FUNCTION_BLOCK FB_FlowLine
(*
********************************************************************************
* Name: FB_Camera
*
* Author:  AutomanH
* Version: 1.0.0
*
* Description:
*	Flow Line Program and motor control
*
* Remarks:
*
*
* Revisions:
*   V1.0.0 -Automanh 2022.06.08
* 	V1.1.0-Automanh 2022.06.20,Add ACT_Motor();
*		V2.0.0-Automanh 2022.07.18 add timeout alarm 
*********************************************************************************)
VAR_INPUT
 arIReachedSensor:ARRAY[1..iColumnsNum] OF BOOL;
 arIVTCCylHPSensor:ARRAY[1..iColumnsNum] OF BOOL;
 arIVTCCylWPSensor:ARRAY[1..iColumnsNum] OF BOOL;
 xIRunningPremit:BOOL;
 xIMotorStop:BOOL;
 xIEmptyDone:BOOL;
 xITryRun:BOOL;
 xIMotorEstop:BOOL;
 xIInit:BOOL;
 xIMotorStartButtonHmi:BOOL;
 xIMotorStopButtonHmi:BOOL;
 xIManualMode:BOOL;
 xIAutoMode:BOOL;
 xIDeviceRunning:BOOL;
END_VAR
VAR_OUTPUT
 arQVTCCylHPValve:ARRAY[1..iColumnsNum] OF BOOL;
 arQVTCCylWPValve:ARRAY[1..iColumnsNum] OF BOOL; 
 xQMotorEstop:BOOL;
 xQMotorStop:BOOL;
 xQMotorStart:BOOL;
 xQBusy:BOOL;
 xQError:BOOL;
 xQDone:BOOL;
END_VAR
VAR
 	//链板线电机启动
 	xMotorStart:BOOL;
	xMotorStop:BOOL;
	// 链板线步骤
	bFlowLineStep: BYTE;
	bFlowLineStepOld:BYTE;
	bMotorCtrlStep:BYTE;
	// 延时
	arTonDelay: ARRAY[1..10] OF ton;
	i:INT;
	_xFirstCycle: BOOL;
	stMotorStatus:DUT_Motor;
	ModeSwitchR_TRIG:R_TRIG;
	MotorStopR_TRIG:R_TRIG;
	InitR_TRIG:R_TRIG;
	bInitStep: BYTE;
	//超时
	tTimeOut:TON;
	
END_VAR
VAR CONSTANT
 	iColumnsNum :INT:=4;
END_VAR

ACT_Motor();
ACT_Flow();
ACT_Manual();
ACT_Init();

ACTION ACT_Flow:


{region "链板线程序"}
tTimeOut(IN:= bFlowLineStepOld =bFlowLineStep AND bFlowLineStepOld<>0,PT:=T#15S , Q=> , ET=> );
IF  tTimeOut.Q THEN
		xQError:=TRUE; 
		tTimeOut(IN:=FALSE); 			
END_IF
	CASE bFlowLineStep OF
	0://启动
		FOR i:=1 TO 10 BY 1 DO
			arTonDelay[i](IN:=FALSE);
		END_FOR
		IF	xIRunningPremit  AND NOT xIEmptyDone  THEN
				bInitStep:=0;
				xMotorStart:=TRUE;
				xMotorStop:=FALSE;
				_xFirstCycle:=TRUE;
				xIRunningPremit:=FALSE;
				xQBusy:=TRUE;
				xQDone:=FALSE;
				bFlowLineStep:=bFlowLineStep +1;
		ELSE
				xMotorStart:=FALSE;
		END_IF
	1://下压气缸回原
		 		bFlowLineStepOld :=bFlowLineStep;
				FOR  i:=1 TO iColumnsNum BY 1 DO
					 arQVTCCylWPValve[i]:=FALSE;
					 arQVTCCylHPValve[i]:=TRUE;
				END_FOR 	
				bFlowLineStep:=bFlowLineStep +1;
	2://判断回原是否完成
		 	bFlowLineStepOld :=bFlowLineStep;
				FOR  i:=1 TO iColumnsNum BY 1 DO
					IF  NOT arIVTCCylHPSensor[i] THEN
						EXIT;	
					 ELSIF  i  =iColumnsNum THEN
							bFlowLineStep:=bFlowLineStep +1;
					 END_IF
				 END_FOR
	3://到位传感器检测
		// bFlowLineStepOld :=bFlowLineStep;
		IF NOT xITryRun THEN
			FOR  i:=1 TO iColumnsNum BY 1 DO
				IF  NOT arIReachedSensor[i]  THEN
					EXIT;
				ELSIF   i =iColumnsNum THEN
					bFlowLineStep:=bFlowLineStep +1;
				END_IF
			END_FOR
		ELSE
				bFlowLineStep:=bFlowLineStep +2;
		END_IF
	4://下压气缸伸出
		 			bFlowLineStepOld :=bFlowLineStep;
					FOR  i:=1 TO iColumnsNum BY 1 DO
							 arQVTCCylWPValve[i]:=TRUE;
							 arQVTCCylHPValve[i]:=FALSE;
					 
					END_FOR
						bFlowLineStep:=bFlowLineStep +1;
	5://检测下压气缸到位
		 		bFlowLineStepOld :=bFlowLineStep;
				bFlowLineStep:=bFlowLineStep +1;
	6://延时1s
		 	bFlowLineStepOld :=bFlowLineStep;
			arTonDelay[3](IN:=TRUE  , PT:=T#1S , Q=> , ET=> );
			IF  	arTonDelay[3].Q THEN
						bFlowLineStep:=bFlowLineStep +1;
						arTonDelay[3](IN:=FALSE);
			END_IF	      
	7://输出链板线Ready信号
		 	bFlowLineStepOld :=bFlowLineStep;
			 xQBusy:=FALSE;
			 xQDone:=TRUE;
			 bFlowLineStep:=0;
	END_CASE
	xIRunningPremit:=FALSE;
{endregion}
END_ACTION

ACTION ACT_Init:
InitR_TRIG(CLK:= xIInit, Q=> );
CASE bInitStep OF
 0:
		IF	InitR_TRIG.Q THEN
				bFlowLineStep:=0;
				xQBusy:=FALSE;
				xQError:=FALSE;
				bFlowLineStepOld:=0;
				bInitStep:=bInitStep +1;
		 END_IF
 1://气缸回原
			FOR  i:=1 TO iColumnsNum BY 1 DO
			 	 arQVTCCylWPValve[i]:=FALSE;
				 arQVTCCylHPValve[i]:=TRUE;
			END_FOR 	
				bInitStep:=bInitStep +1;
 2://链板线停止
 			xQMotorEstop:=FALSE;
		  xQMotorStop:=FALSE;
		  xQMotorStart:=FALSE;
			xQBusy:=FALSE;
			bInitStep:=0;
END_CASE
xIInit:=FALSE;
END_ACTION

ACTION ACT_Manual:
IF  (xMotorStart AND  xIDeviceRunning )  OR
 		(xIMotorStartButtonHmi AND xIManualMode) THEN
				xMotorStart:=TRUE;
				xMotorStop:=FALSE;
ELSIF
 	 (xIMotorStop AND  xIDeviceRunning )  OR
 	(xIMotorStopButtonHmi AND xIManualMode)	THEN
			xMotorStart:=FALSE;
			xMotorStop:=TRUE;
END_IF
END_ACTION

ACTION ACT_Motor:
ModeSwitchR_TRIG(CLK:= xIManualMode (*XOR xIAutoMode*) , Q=> );
CASE  bMotorCtrlStep  OF
0://等待激活
			IF   xIMotorEstop THEN
			 		bMotorCtrlStep:=1;
			ELSIF xMotorStop	 THEN
			 		bMotorCtrlStep:=2;
			ELSIF ModeSwitchR_TRIG.Q THEN
			 		bMotorCtrlStep:=4;
			ELSIF xMotorStart	 THEN
			 		bMotorCtrlStep:=3;
			END_IF
1://急停被拍下
		xQMotorEstop:=TRUE;
		xQMotorStart:=FALSE;
		bMotorCtrlStep:=0;
2://停止被按下
		xQMotorStart:=FALSE;
		xQMotorStop:=TRUE;
		bMotorCtrlStep:=0;
3://启动被按下
			xQMotorStop:=FALSE;
			xQMotorStart:=TRUE;
			bMotorCtrlStep:=0;
4://设备模式切换
			xQMotorStart:=FALSE;
			xQMotorStop:=TRUE;
			bMotorCtrlStep:=0;
			bFlowLineStep:=0;
END_CASE
END_ACTION

END_FUNCTION_BLOCK

(* stored: Version 1.1.0.1, ProductVersion 3.1.4024.9
   POU FB_FlowLine: Id {52997166-3b63-4e55-9278-d93ff937da70}, SpecialFunc None
   Action ACT_Flow: Id {8a8dac4c-17a0-452b-be41-4bef968f9fe3}
   Action ACT_Init: Id {6524b2a2-a9d5-4f5a-8fad-02d8e90a8192}
   Action ACT_Manual: Id {be38eeb0-0032-4be1-8538-9852e13dc970}
   Action ACT_Motor: Id {849b814a-2f32-478a-9aea-f75e9105b6dc} *)
